KUKA KRL program: style1app1opt3B.src, style1app1opt3B.dat

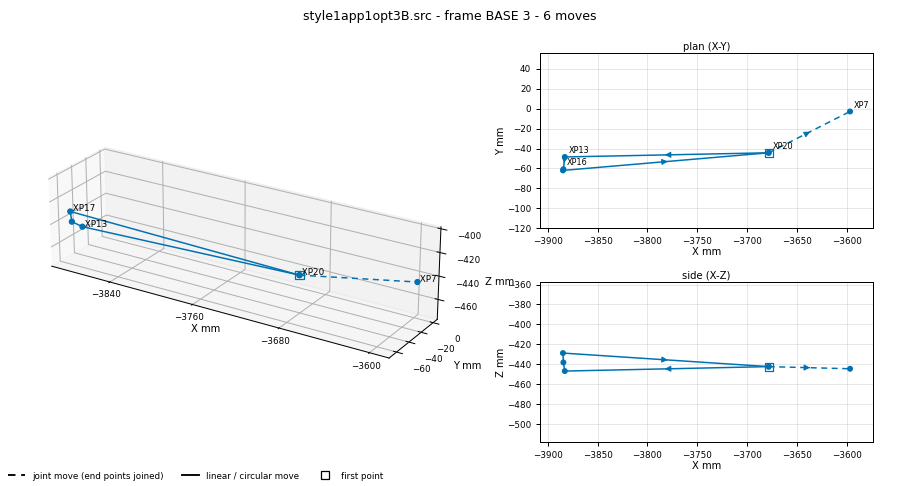
[picture p0: tool path of style1app1opt3B.src in frame BASE 3, 6 of 6 moves have a stored position in this frame; points joined in program order, loops and branches not executed]
--- style1app1opt3B.src ---
&ACCESS RVO1
&REL 227
&COMMENT 03-10-R1 PNW1 NUT 3 ST2
&PARAM EDITMASK = *
&PARAM TEMPLATE = C:\KRC\TP\Nutweld\Template\NutWeld_Vorgabe
&PARAM DISKPATH = KRC:\R1\Program\StyleApps\Options
DEF style1app1opt3B( )
   ;FOLD INI
      ;FOLD BASISTECH INI
         GLOBAL INTERRUPT DECL 3 WHEN $STOPMESS==TRUE DO IR_STOPM ( )
         INTERRUPT ON 3
         BAS (#INITMOV,0 )
      ;ENDFOLD (BASISTECH INI)
      ;FOLD NutWeld
      ;ENDFOLD (NutWeld)
      ;FOLD USER INI
         ;Make your modifications here

      ;ENDFOLD (USER INI)
   ;ENDFOLD (INI)
;********************************
; Gestamp Standards
; Line - BMW G65 (cell 03)
; Robot 03-10-R1 (BMW-03-10-R1-PNW1)
; Application - WELD NUT 3 (PN3) AT THE CENTERLINE PEDESTAL - PART FROM PICKUP 2 (B)
;********************************
; CALLED BY Style1Opt1. APPROACH THE PEDESTAL (BASE 3 "NUT WELDER"), WAIT FOR THE NUT PRELOAD
; (NEXT_NUT_READY), MOVE THE PART TO THE WELD POSITION P16, WELD WITH CENTERLINE_WELD (NOT IN DRY
; CYCLE), LEAVE THE PEDESTAL.
;WARNING: BEFORE THE ROBOT MOVES IN, GUN OPEN, SUBMIT AND WATER ARE CHECKED (GUN_OPEN_CHECK) -
;  NOT CLAMP OPEN OR QFP RETURNED (F01)
;NOTE: THE PEDESTAL MOVES MIX BASE MODE AND EXTERNAL-TCP MODE (extTCP); THE WELD POSITION
;  P16 IS TAUGHT IN BASE MODE (F22)

;APPROACH THE PEDESTAL - P20
;FOLD LIN P20 CONT Vel=2 m/s CPDAT6 Tool[1]:TOOL 1 Base[3]:NUT WELDER extTCP;%{PE}%R 8.3.43,%MKUKATPBASIS,%CMOVE,%VLIN,%P 1:LIN, 2:P20, 3:C_DIS C_DIS, 5:2, 7:CPDAT6
$BWDSTART=FALSE
LDAT_ACT=LCPDAT6
FDAT_ACT=FP20
BAS(#CP_PARAMS,2)
LIN XP20 C_DIS C_DIS
;ENDFOLD
;GUN MONITORING - INTERRUPTS 20-22 CALL GUN_OPEN_LOST (BRAKE F, QUIT MESSAGE) WHEN THE GUN LEAVES THE
;OPEN RANGE (CL_GunStrokePositionLPT 137000..142000) OR THE SUBMIT STOPS WHILE THE ROBOT MOVES INTO
;OR OUT OF THE PEDESTAL. EDGE TRIGGERED: GUN_OPEN_CHECK CONFIRMS THE GUN OPEN AFTER EVERY ON (F01)
;WARNING: THE RANGE IS WRITTEN HERE AS LITERALS; KEEP IT EQUAL TO nGunOpenMin/nGunOpenMax IN
;  GUN_OPEN_CHECK.dat (F01)
INTERRUPT DECL 20 WHEN CL_GunStrokePositionLPT<137000 DO GUN_OPEN_LOST()
INTERRUPT DECL 21 WHEN CL_GunStrokePositionLPT>142000 DO GUN_OPEN_LOST()
INTERRUPT DECL 22 WHEN $PRO_STATE0<>#P_ACTIVE DO GUN_OPEN_LOST()
;CYCLE-TIME MEASUREMENT (NO EFFECT ON THE SEQUENCE): ROBOT STOPPED AT THE WAIT POINT (WAIT SEC 0),
;$TIMER[20] FROM HERE FOR NUT 3 (CL_CYCLE_TIME, F52)
WAIT SEC 0
CL_CYCLE_START(3)
;WAIT NUT PRELOADED - NEXT_NUT_READY (SET WHEN THE PRELOAD ENDS, QFP SEEN RETURNED; NO NUT SENSOR,
;  F13)
;NOTE: NO TIMEOUT, NO MESSAGE (F15). IN DRY CYCLE NOTHING SETS IT: THE CYCLE HANGS HERE (F04)
WAIT FOR NEXT_NUT_READY==TRUE
;CYCLE-TIME MARK - STEP 1 NUT READY (CL_CYCLE_TIME, F52)
CL_CYCLE_TIME(1)
;GUN MONITORING ON FIRST (THE INTERRUPTS FIRE ONLY ON A CHANGE), THEN THE INTERLOCK: GUN OPEN,
;SUBMIT RUNNING, WATER OK (GUN_OPEN_CHECK); THE MONITORING STAYS ON WHILE THE ROBOT MOVES IN (F01)
INTERRUPT ON 20
INTERRUPT ON 21
INTERRUPT ON 22
GUN_OPEN_CHECK()
;MOVE IN - P13 (2 M/S), THEN THE WELD POSITION P16 OUTSIDE DRY CYCLE
;FOLD LIN P13 CONT Vel=2 m/s CPDAT4 Tool[1]:TOOL 1 Base[3]:NUT WELDER extTCP;%{PE}%R 8.3.43,%MKUKATPBASIS,%CMOVE,%VLIN,%P 1:LIN, 2:P13, 3:C_DIS C_DIS, 5:2, 7:CPDAT4
$BWDSTART=FALSE
LDAT_ACT=LCPDAT4
FDAT_ACT=FP13
BAS(#CP_PARAMS,2)
LIN XP13 C_DIS C_DIS
;ENDFOLD

;OUTSIDE DRY CYCLE ONLY (SIGNAL $IN[4] di004UseDryCycle OFF): WELD POSITION P16 AND CENTERLINE_WELD()
;NOTE: $IN[4] IS RE-READ AT EVERY STEP; SWITCHED ON MID-CYCLE, THIS NUT IS NOT WELDED AND
;  THE PART CAN STILL REACH THE GOOD DROP (F05)
IF NOT di004UseDryCycle THEN
;FOLD LIN P16 Vel=2 m/s CPDAT11 Tool[1]:TOOL 1 Base[3]:NUT WELDER;%{PE}%R 8.3.43,%MKUKATPBASIS,%CMOVE,%VLIN,%P 1:LIN, 2:P16, 3:, 5:2, 7:CPDAT11
$BWDSTART=FALSE
LDAT_ACT=LCPDAT11
FDAT_ACT=FP16
BAS(#CP_PARAMS,2)
LIN XP16
;ENDFOLD
;ROBOT AT THE WELD POSITION (WAIT SEC 0 STOPS THE ADVANCE RUN): GUN MONITORING OFF, THE GUN
;CLOSES ON PURPOSE IN CENTERLINE_WELD
WAIT SEC 0
INTERRUPT OFF 20
INTERRUPT OFF 21
INTERRUPT OFF 22
;NUT WELD AT THE PEDESTAL (CENTERLINE_WELD: CLAMP, GUN, INTENSIFY, BOSCH WELD, GUN OPEN)
CENTERLINE_WELD()
;GUN MONITORING ON WHILE LEAVING, THEN THE GUN OPEN IS CONFIRMED AGAIN (GUN_OPEN_CHECK): A GUN THAT
;LEFT THE OPEN RANGE AFTER THE CHECK INSIDE CENTERLINE_WELD WOULD NOT TRIGGER THE INTERRUPTS (F01)
INTERRUPT ON 20
INTERRUPT ON 21
INTERRUPT ON 22
GUN_OPEN_CHECK()
ENDIF
;LEAVE THE PEDESTAL - P17, P20, P7 (60 %) (THE DRY CYCLE CONTINUES HERE)
;FOLD LIN P17 Vel=2 m/s CPDAT12 Tool[1]:TOOL 1 Base[3]:NUT WELDER;%{PE}%R 8.3.43,%MKUKATPBASIS,%CMOVE,%VLIN,%P 1:LIN, 2:P17, 3:, 5:2, 7:CPDAT12
$BWDSTART=FALSE
LDAT_ACT=LCPDAT12
FDAT_ACT=FP17
BAS(#CP_PARAMS,2)
LIN XP17
;ENDFOLD
;ROBOT OUT OF THE PEDESTAL (WAIT SEC 0 STOPS THE ADVANCE RUN, NO APPROXIMATION HERE): GUN
;MONITORING OFF
WAIT SEC 0
INTERRUPT OFF 20
INTERRUPT OFF 21
INTERRUPT OFF 22
;FOLD LIN P20 Vel=2 m/s CPDAT10 Tool[1]:TOOL 1 Base[3]:NUT WELDER extTCP;%{PE}%R 8.3.43,%MKUKATPBASIS,%CMOVE,%VLIN,%P 1:LIN, 2:P20, 3:, 5:2, 7:CPDAT10
$BWDSTART=FALSE
LDAT_ACT=LCPDAT10
FDAT_ACT=FP20
BAS(#CP_PARAMS,2)
LIN XP20
;ENDFOLD
;LAST NUT OF THE PART: NO NEXT NUT IS REQUESTED HERE (THE NEXT PICK STARTS THE PRELOAD)
;FOLD PTP P7 Vel=60 % PDAT25 Tool[1]:TOOL 1 Base[3]:NUT WELDER extTCP;%{PE}%R 8.3.43,%MKUKATPBASIS,%CMOVE,%VPTP,%P 1:PTP, 2:P7, 3:, 5:60, 7:PDAT25
$BWDSTART=FALSE
PDAT_ACT=PPDAT25
FDAT_ACT=FP7
BAS(#PTP_PARAMS,60)
PTP XP7
;ENDFOLD


END

--- style1app1opt3B.dat ---
&ACCESS RVO1
&REL 227
&COMMENT GE4_003_GUN1
&PARAM EDITMASK = *
&PARAM TEMPLATE = C:\KRC\TP\Nutweld\Template\NutWeld_Vorgabe
&PARAM DISKPATH = KRC:\R1\Program\StyleApps\Options
DEFDAT  style1app1opt3B
;FOLD EXTERNAL DECLARATIONS;%{PE}%MKUKATPBASIS,%CEXT,%VCOMMON,%P
;FOLD BASISTECH EXT;%{PE}%MKUKATPBASIS,%CEXT,%VEXT,%P
EXT  BAS (BAS_COMMAND  :IN,REAL  :IN )
;ENDFOLD (BASISTECH EXT)
;FOLD NutWeld
;ENDFOLD (NutWeld)
;FOLD USER EXT;%{E}%MKUKATPUSER,%CEXT,%VEXT,%P
;Make here your modifications
;ENDFOLD (USER EXT)
DECL E6POS XP20={X -3678.25781,Y -44.2650108,Z -442.362579,A -178.367340,B 0.267035842,C 179.968063,S 2,T 2,E1 0.0,E2 0.0,E3 0.0,E4 0.0,E5 0.0,E6 0.0}
DECL FDAT FP20={TOOL_NO 1,BASE_NO 3,IPO_FRAME #TCP,POINT2[] " ",TQ_STATE FALSE}
;ENDFOLD (EXTERNAL DECLARATIONS)
DECL FDAT FPNW1={TOOL_NO 1,BASE_NO 3,IPO_FRAME #TCP,POINT2[] " ",TQ_STATE FALSE}
DECL E6POS XPNW1={X -684.340210,Y -936.680359,Z 6.96372366,A -85.0124512,B -3.00309157,C -5.37728167,S 2,T 11,E1 0.0,E2 0.0,E3 0.0,E4 0.0,E5 0.0,E6 0.0}
DECL BASIS_SUGG_T LAST_BASIS={POINT1[] "P18                     ",POINT2[] "P18                     ",CP_PARAMS[] "CPDAT0                  ",PTP_PARAMS[] "PDAT26                  ",CONT[] "                        ",CP_VEL[] "2                       ",PTP_VEL[] "100                     ",SYNC_PARAMS[] "SYNCDAT                 ",SPL_NAME[] "S0                      ",A_PARAMS[] "ADAT0                   "}
DECL NutWeld_SUGG_T LAST_NutWeld={POINT1[] "PNW3_SPOT03             ",POINT2[] "PNW0                    ",CP_PARAMS[] "CPDATNutWeld0           ",PTP_PARAMS[] "PDATNutWeld0            ",CONT[] "C_PTP                   ",CP_VEL[] "2                       ",PTP_VEL[] "100                     ",SYNC_PARAMS[] "SYNCDAT                 ",SPL_NAME[] "S0                      ",NutWeld_PARAMS[] "NutData3_3              ",GunNr 3,SpotNr 3,Offset 10}
DECL MODULEPARAM_T LAST_TP_PARAMS={PARAMS[] "NutWeld_CmdPos=Weld; NutWeld_Move=LIN; NutWeld_NutWeldDat=NutWeldDAT1; NutWeld_NWGunNr=3; NutWeld_NWSpotNr=3; NutWeld_NWOffset=0; Kuka.MoveDataName=CPDAT2; Kuka.VelocityPath=2; Kuka.PointName=PNW1; Kuka.BlendingEnabled=False; Kuka.FrameData.tq_state=False; Kuka.FrameData.base_no=3; Kuka.FrameData.tool_no=1; Kuka.FrameData.ipo_frame=#TCP; Kuka.FrameData.point2=; Kuka.MovementData.apo_fac=50; Kuka.MovementData.apo_dist=100; Kuka.MovementData.axis_acc=100; Kuka.MovementData.axis_vel=100; Kuka.MovementData.circ_typ=#BASE; Kuka.MovementData.exax_ign=0; Kuka.MovementData.jerk_fac=50; Kuka.MovementData.ori_typ=#VAR; Kuka.MovementData.acc=100; Kuka.MovementData.gear_jerk=50    "}
DECL LDAT Lpnw1={VEL 2.00000,ACC 100.000,APO_DIST 100.000,APO_FAC 50.0000,AXIS_VEL 100.000,AXIS_ACC 100.000,ORI_TYP #VAR,CIRC_TYP #BASE,JERK_FAC 50.0000,GEAR_JERK 50.0000,EXAX_IGN 0}
DECL E6POS XP7={X -3596.62695,Y -2.77881479,Z -444.531586,A -178.368134,B 0.266892016,C 179.968369,S 2,T 34,E1 0.0,E2 0.0,E3 0.0,E4 0.0,E5 0.0,E6 0.0}
DECL FDAT FP7={TOOL_NO 1,BASE_NO 3,IPO_FRAME #TCP,POINT2[] " ",TQ_STATE FALSE}
DECL E6POS XP13={X -3882.93384,Y -48.4484138,Z -446.836792,A -178.367340,B 0.267035872,C 179.968063,S 2,T 2,E1 0.0,E2 0.0,E3 0.0,E4 0.0,E5 0.0,E6 0.0}
DECL FDAT FP13={TOOL_NO 1,BASE_NO 3,IPO_FRAME #TCP,POINT2[] " ",TQ_STATE FALSE}
DECL LDAT LCPDAT4={VEL 2.00000,ACC 100.000,APO_DIST 2.00000,APO_FAC 50.0000,AXIS_VEL 100.000,AXIS_ACC 100.000,ORI_TYP #VAR,CIRC_TYP #BASE,JERK_FAC 50.0000,GEAR_JERK 50.0000,EXAX_IGN 0}
DECL PDAT PPDAT25={VEL 100.000,ACC 100.000,APO_DIST 100.000,APO_MODE #CDIS,GEAR_JERK 50.0000,EXAX_IGN 0}
DECL LDAT LCPDAT6={VEL 2.00000,ACC 100.000,APO_DIST 2.00000,APO_FAC 50.0000,AXIS_VEL 100.000,AXIS_ACC 100.000,ORI_TYP #VAR,CIRC_TYP #BASE,JERK_FAC 50.0000,GEAR_JERK 50.0000,EXAX_IGN 0}
DECL LDAT LCPDAT10={VEL 2.00000,ACC 100.000,APO_DIST 100.000,APO_FAC 50.0000,AXIS_VEL 100.000,AXIS_ACC 100.000,ORI_TYP #VAR,CIRC_TYP #BASE,JERK_FAC 50.0000,GEAR_JERK 50.0000,EXAX_IGN 0}
DECL E6POS XP16={X -3884.36157,Y -60.7767830,Z -438.167816,A -178.367172,B -0.266017556,C 179.960464,S 2,T 2,E1 0.0,E2 0.0,E3 0.0,E4 0.0,E5 0.0,E6 0.0}
DECL FDAT FP16={TOOL_NO 1,BASE_NO 3,IPO_FRAME #BASE,POINT2[] " ",TQ_STATE FALSE}
DECL LDAT LCPDAT11={VEL 2.00000,ACC 100.000,APO_DIST 100.000,APO_FAC 50.0000,AXIS_VEL 100.000,AXIS_ACC 100.000,ORI_TYP #VAR,CIRC_TYP #BASE,JERK_FAC 50.0000,GEAR_JERK 50.0000,EXAX_IGN 0}
DECL E6POS XP17={X -3884.77832,Y -61.9626274,Z -428.770508,A -178.367172,B -0.266017497,C 179.960464,S 2,T 2,E1 0.0,E2 0.0,E3 0.0,E4 0.0,E5 0.0,E6 0.0}
DECL FDAT FP17={TOOL_NO 1,BASE_NO 3,IPO_FRAME #BASE,POINT2[] " ",TQ_STATE FALSE}
DECL LDAT LCPDAT12={VEL 2.00000,ACC 100.000,APO_DIST 100.000,APO_FAC 50.0000,AXIS_VEL 100.000,AXIS_ACC 100.000,ORI_TYP #VAR,CIRC_TYP #BASE,JERK_FAC 50.0000,GEAR_JERK 50.0000,EXAX_IGN 0}
ENDDAT
